INTERFACE I_JsonPath

METHOD PUBLIC TryRead : HRESULT
VAR_INPUT
	Path : T_MaxString;
	Destination : ANY;
END_VAR
END_METHOD

END_INTERFACE

(* stored: Version 1.1.0.1, ProductVersion 3.1.4024.12
   Itf I_JsonPath: Id {099780fc-16fb-4ca3-b4ec-a59f8599d9b7}
   Method TryRead: Id {9c1139bf-eae3-4f48-b33d-605dfa2e97d2} *)
